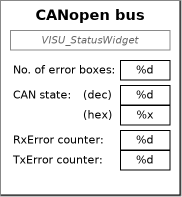
VISUALIZATION VISU_CANopenBus  // 182x197
VAR_IN_OUT
	ref : CANopenBus;
	widget : CANopenBusWidget;
END_VAR
    Rectangle (0,0 180x195)
    Rectangle (0,0 180x30), "CANopen bus"
    Label (10,55 135x30), "No. of error boxes:"
    Rectangle (120,60 50x20), "%d", text variable: ref.error
    Frame (10,30 160x20)
        shows VISU_StatusWidget(widget := widget.actualStatus)
    Label (10,80 155x30), "CAN state:"
    Rectangle (120,85 50x20), "%d", text variable: ref.canState
    Label (80,85 35x20), "(dec)"
    Rectangle (120,105 50x20), "%x", text variable: ref.canState
    Label (80,105 40x20), "(hex)"
    Label (10,125 135x30), "RxError counter:"
    Rectangle (120,130 50x20), "%d", text variable: ref.rxErrorCounter
    Label (10,145 135x30), "TxError counter:"
    Rectangle (120,150 50x20), "%d", text variable: ref.txErrorCounter
END_VISUALIZATION

(* stored: Version 1.1.0.1, ProductVersion 3.1.4019.2
   Visu VISU_CANopenBus: Id {6f6441ac-cf67-441c-a381-02b6cfe86442} *)
